{attribute 'strict'}
TYPE MoverState_enum :
(
	MV_IDLE				:= 0,
	MV_RESET			:= 10,
	MV_M1_READMODE		:= 20,
	MV_M1_EVALMODE		:= 30,
	MV_M1_READSTATUS	:= 40,
	MV_M1_EVALSTATUS	:= 50,
	MV_M1_DETECT		:= 60,
	MV_ENABLING			:= 70,
	MV_ADDTOGROUP		:= 80,
	MV_READGROUPSTATUS	:= 90,
	MV_ENABLEGROUP		:= 100,
	MV_RUN				:= 110,
	MV_STOPPING			:= 120,
	MV_DISABLING		:= 130,
	MV_ERROR			:= 140
);
END_TYPE

(* stored: Version 1.1.0.1, ProductVersion 3.1.4024.9
   DUT MoverState_enum: Id {89a812d1-f23a-47af-b019-1e4ee25dac44} *)
